FUNCTION_BLOCK FB_Motor_run_time
VAR_INPUT
	Start:BOOL;
	Reset:BOOL;
END_VAR
VAR_OUTPUT
	Hours:REAL;
	Minutes:REAL;
	Sec:REAL;
END_VAR
VAR
	T2_dn:BOOL;
	one_sec_pulse:BOOL;
	Min_pulse:BOOL;
	Hour_pulse:BOOL;
	End_pulse:BOOL;
	TON_0: TON;
	TON_1: TON;
	R_TRIG_0: R_TRIG;
	CTU_0: CTU;
	R_TRIG_1: R_TRIG;
	R_TRIG_2: R_TRIG;
	CTU_1: CTU;
	CTU_2: CTU;
END_VAR

M_Main();

METHOD M_Main
VAR_INPUT
END_VAR
VAR_INST // added by the converter: edge detectors and wires of the graphical bodies
    _w1, _w2 : ANY;
END_VAR
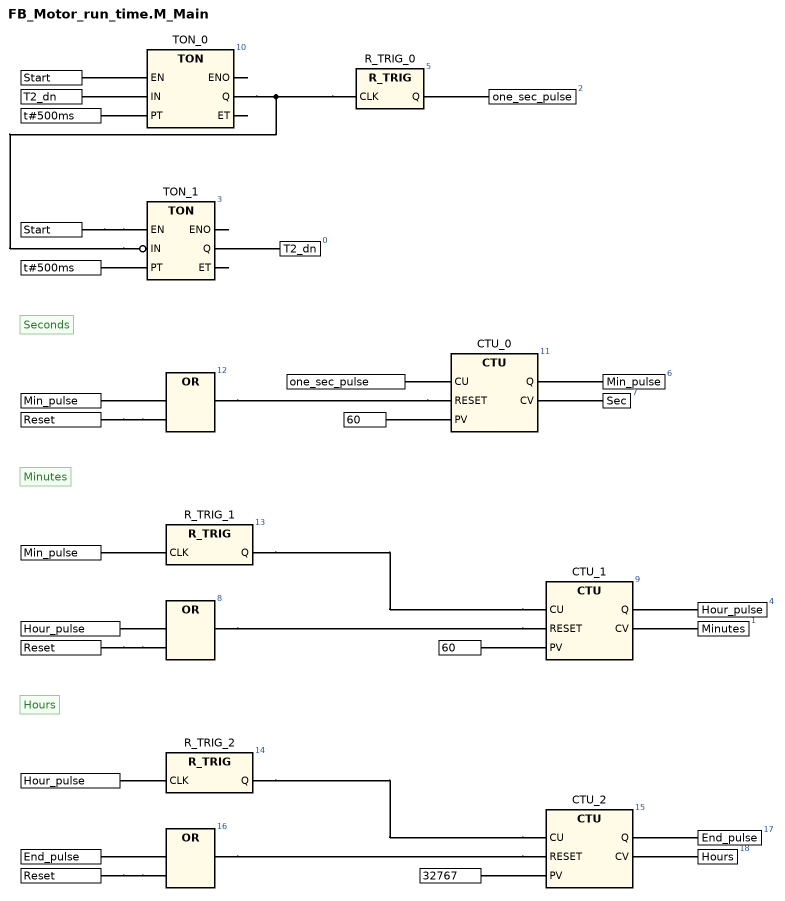
T2_dn := TON_1.Q;
Minutes := CTU_1.CV;
one_sec_pulse := R_TRIG_0.Q;
IF Start THEN
    TON_1(IN := NOT TON_0.Q, PT := t#500ms); // TON
END_IF
Hour_pulse := CTU_1.Q;
R_TRIG_0(CLK := TON_0.Q); // R_TRIG
Min_pulse := CTU_0.Q;
Sec := CTU_0.CV;
CTU_1(CU := R_TRIG_1.Q, RESET := Hour_pulse OR Reset, PV := 60); // CTU
IF Start THEN
    TON_0(IN := T2_dn, PT := t#500ms); // TON
END_IF
CTU_0(CU := one_sec_pulse, RESET := _w1, PV := 60); // CTU
// Seconds
_w1 := Min_pulse OR Reset;
// Minutes
R_TRIG_1(CLK := Min_pulse); // R_TRIG
// Hours
R_TRIG_2(CLK := Hour_pulse); // R_TRIG
CTU_2(CU := R_TRIG_2.Q, RESET := _w2, PV := 32767); // CTU
_w2 := End_pulse OR Reset;
End_pulse := CTU_2.Q;
Hours := CTU_2.CV;
END_METHOD

END_FUNCTION_BLOCK

(* stored: Version 1.1.0.1, ProductVersion 3.1.4024.0
   POU FB_Motor_run_time: Id {b918734f-a0bb-4f45-861e-888b13a12d1e}, SpecialFunc None
   Method M_Main: Id {051e9868-6516-46dd-97e8-c3bdc28daf72} *)
